(* PLC project Unnamed, Unknown Unnamed 1 *)
(* stored: creationDateTime 2024-12-05T23:43:34, modificationDateTime 2024-12-05T23:56:35 *)

PROGRAM GrabTheApple
  VAR
    CLAW_LEFT : BOOL;
    CLAW_RIGHT : BOOL;
    CLAW_GRAB : BOOL;
    APPLE_EXISTS : BOOL;
    APPLE_IS_LEFT : BOOL;
    APPLE_IS_RIGHT : BOOL;
  END_VAR

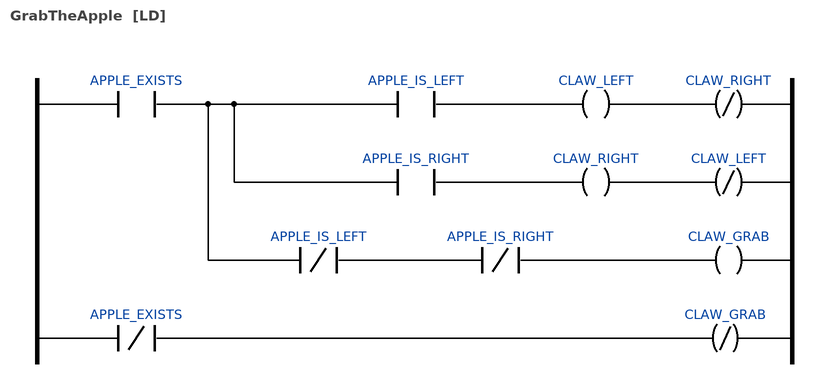
(* LD diagram, written out as Structured Text *)
CLAW_LEFT := APPLE_EXISTS AND APPLE_IS_LEFT;
CLAW_RIGHT := NOT (APPLE_EXISTS AND APPLE_IS_LEFT);
CLAW_LEFT := NOT (APPLE_EXISTS AND APPLE_IS_RIGHT);
CLAW_RIGHT := APPLE_EXISTS AND APPLE_IS_RIGHT;
CLAW_GRAB := APPLE_EXISTS AND NOT APPLE_IS_LEFT AND NOT APPLE_IS_RIGHT;
CLAW_GRAB := NOT (NOT APPLE_EXISTS);
END_PROGRAM

CONFIGURATION Config0
  RESOURCE Res0 ON PLC
    TASK task0(INTERVAL := T#20ms, PRIORITY := 0);
    PROGRAM instance0 WITH task0 : GrabTheApple;
  END_RESOURCE
END_CONFIGURATION
